PROGRAM Kommunikation_UDP
VAR
	Connect			:FB_SocketUdpCreate;
	Send			:FB_SocketUdpSendTo;
	Receive			:FB_SocketUdpReceiveFrom;
	
	Connect_		:FB_SocketConnect;
	Send_			:FB_SocketSend;
END_VAR

VAR_INPUT
	Receive_		:FB_SocketReceive;
END_VAR

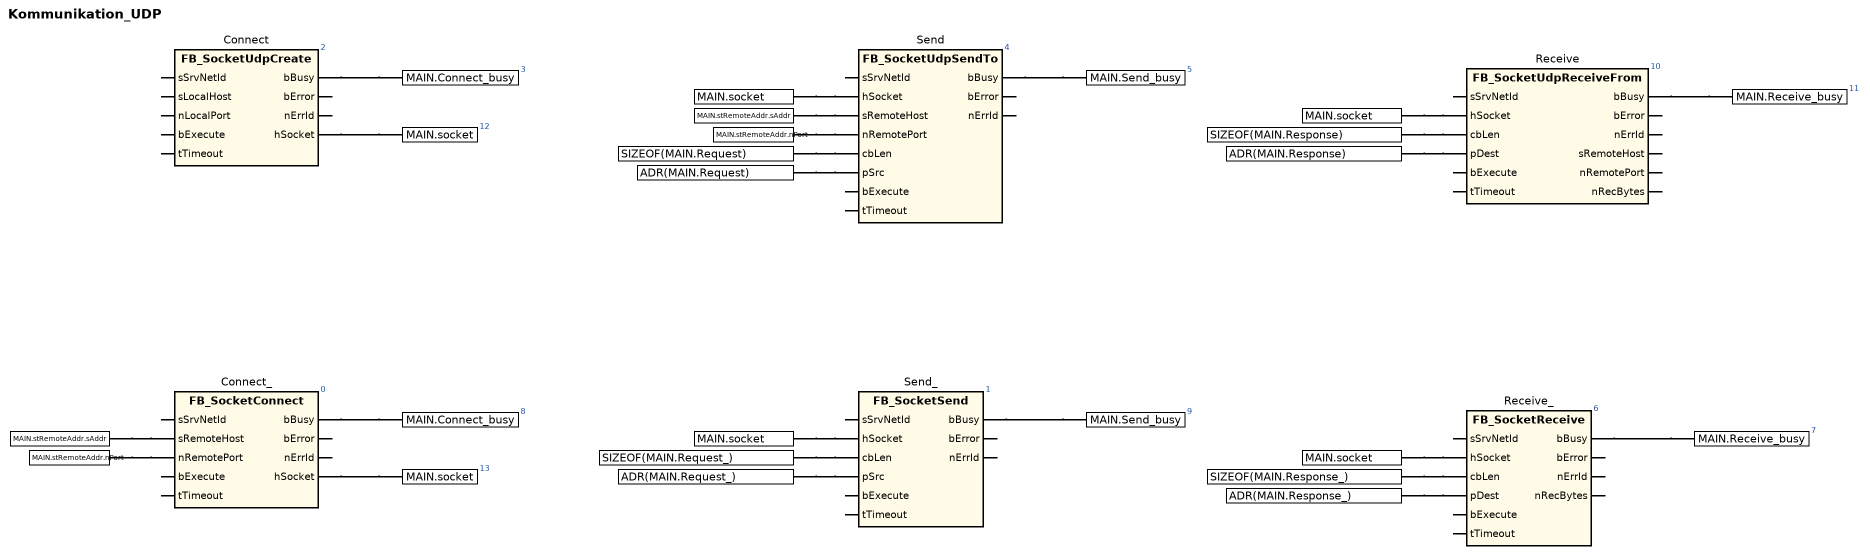
Connect_(sRemoteHost := MAIN.stRemoteAddr.sAddr, nRemotePort := MAIN.stRemoteAddr.nPort); // FB_SocketConnect
Send_(hSocket := MAIN.socket, cbLen := SIZEOF(MAIN.Request_), pSrc := ADR(MAIN.Request_)); // FB_SocketSend
Connect(); // FB_SocketUdpCreate
MAIN.Connect_busy := Connect.bBusy;
Send(
    hSocket := MAIN.socket,
    sRemoteHost := MAIN.stRemoteAddr.sAddr,
    nRemotePort := MAIN.stRemoteAddr.nPort,
    cbLen := SIZEOF(MAIN.Request),
    pSrc := ADR(MAIN.Request)); // FB_SocketUdpSendTo
MAIN.Send_busy := Send.bBusy;
Receive_(hSocket := MAIN.socket, cbLen := SIZEOF(MAIN.Response_), pDest := ADR(MAIN.Response_)); // FB_SocketReceive
MAIN.Receive_busy := Receive_.bBusy;
MAIN.Connect_busy := Connect_.bBusy;
MAIN.Send_busy := Send_.bBusy;
Receive(hSocket := MAIN.socket, cbLen := SIZEOF(MAIN.Response), pDest := ADR(MAIN.Response)); // FB_SocketUdpReceiveFrom
MAIN.Receive_busy := Receive.bBusy;
MAIN.socket := Connect.hSocket;
MAIN.socket := Connect_.hSocket;

END_PROGRAM

(* stored: Version 1.1.0.1
   POU Kommunikation_UDP: Id {a70d75a6-6c63-4c56-922d-2334b211690b}, SpecialFunc None *)
